// TIA Portal V21 export
ORGANIZATION_BLOCK "Date_Time_Block"   // OB200, LAD, ProgramCycle
{ S7_Optimized_Access := 'TRUE' }
// stored: SetENOAutomatically false
   VAR_TEMP   // added for the SCL form of the ladder/FBD networks
      _w1 : Bool;
      _w2 : Bool;
      _w3 : Bool;
   END_VAR
BEGIN

REGION Network 1: Convert Date to String
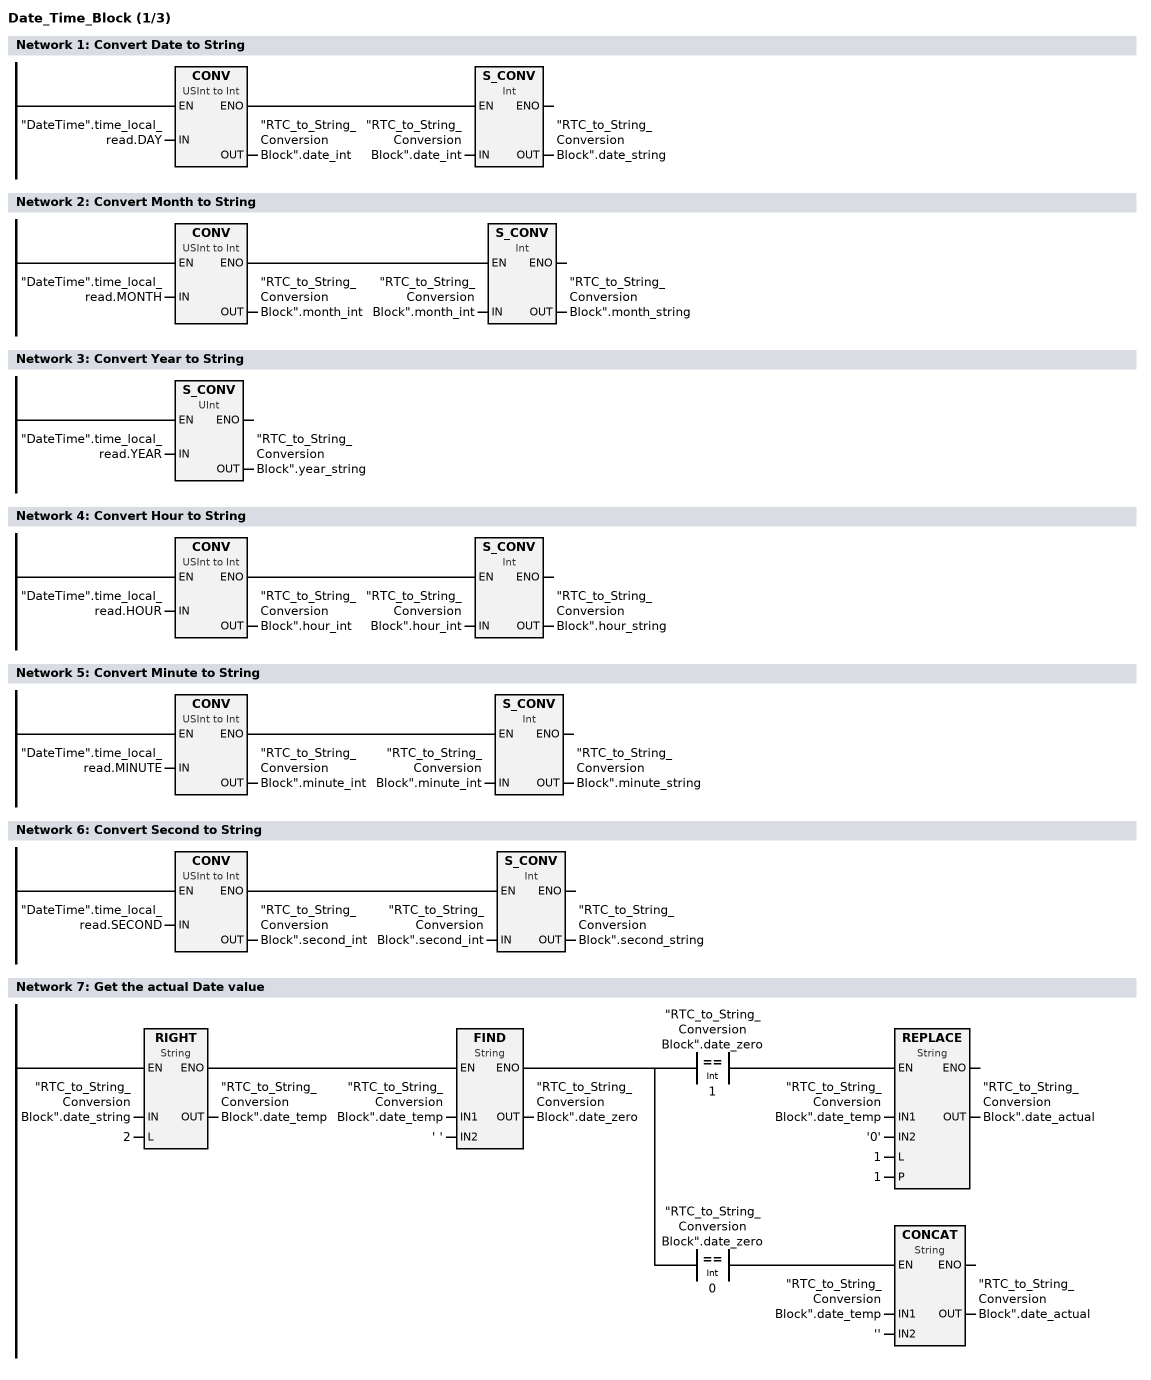
   RUNG wire#powerrail
      { S7_Templates := "[SrcType := USInt, DestType := Int]"; S7_GenerateENO := "TRUE" } Convert(in := "DateTime".time_local_read.DAY, out => "RTC_to_String_Conversion Block".date_int)
      { S7_Templates := "[src_type := Int, dest_type := String]" } S_CONV(IN := "RTC_to_String_Conversion Block".date_int, OUT => "RTC_to_String_Conversion Block".date_string)
   END_RUNG
   // the same network as SCL:
   // ENO of a box is taken as its EN; it also drops when the box reports an error
   "RTC_to_String_Conversion Block".date_int := USINT_TO_INT("DateTime".time_local_read.DAY);
   S_CONV(IN := "RTC_to_String_Conversion Block".date_int, OUT => "RTC_to_String_Conversion Block".date_string);
END_REGION

REGION Network 2: Convert Month to String
   RUNG wire#powerrail
      { S7_Templates := "[SrcType := USInt, DestType := Int]"; S7_GenerateENO := "TRUE" } Convert(in := "DateTime".time_local_read.MONTH, out => "RTC_to_String_Conversion Block".month_int)
      { S7_Templates := "[src_type := Int, dest_type := String]" } S_CONV(IN := "RTC_to_String_Conversion Block".month_int, OUT => "RTC_to_String_Conversion Block".month_string)
   END_RUNG
   // the same network as SCL:
   // ENO of a box is taken as its EN; it also drops when the box reports an error
   "RTC_to_String_Conversion Block".month_int := USINT_TO_INT("DateTime".time_local_read.MONTH);
   S_CONV(IN := "RTC_to_String_Conversion Block".month_int,
          OUT => "RTC_to_String_Conversion Block".month_string);
END_REGION

REGION Network 3: Convert Year to String
   RUNG wire#powerrail
      { S7_Templates := "[src_type := UInt, dest_type := String]" } S_CONV(IN := "DateTime".time_local_read.YEAR, OUT => "RTC_to_String_Conversion Block".year_string)
   END_RUNG
   // the same network as SCL:
   S_CONV(IN := "DateTime".time_local_read.YEAR, OUT => "RTC_to_String_Conversion Block".year_string);
END_REGION

REGION Network 4: Convert Hour to String
   RUNG wire#powerrail
      { S7_Templates := "[SrcType := USInt, DestType := Int]"; S7_GenerateENO := "TRUE" } Convert(in := "DateTime".time_local_read.HOUR, out => "RTC_to_String_Conversion Block".hour_int)
      { S7_Templates := "[src_type := Int, dest_type := String]" } S_CONV(IN := "RTC_to_String_Conversion Block".hour_int, OUT => "RTC_to_String_Conversion Block".hour_string)
   END_RUNG
   // the same network as SCL:
   // ENO of a box is taken as its EN; it also drops when the box reports an error
   "RTC_to_String_Conversion Block".hour_int := USINT_TO_INT("DateTime".time_local_read.HOUR);
   S_CONV(IN := "RTC_to_String_Conversion Block".hour_int, OUT => "RTC_to_String_Conversion Block".hour_string);
END_REGION

REGION Network 5: Convert Minute to String
   RUNG wire#powerrail
      { S7_Templates := "[SrcType := USInt, DestType := Int]"; S7_GenerateENO := "TRUE" } Convert(in := "DateTime".time_local_read.MINUTE, out => "RTC_to_String_Conversion Block".minute_int)
      { S7_Templates := "[src_type := Int, dest_type := String]" } S_CONV(IN := "RTC_to_String_Conversion Block".minute_int, OUT => "RTC_to_String_Conversion Block".minute_string)
   END_RUNG
   // the same network as SCL:
   // ENO of a box is taken as its EN; it also drops when the box reports an error
   "RTC_to_String_Conversion Block".minute_int := USINT_TO_INT("DateTime".time_local_read.MINUTE);
   S_CONV(IN := "RTC_to_String_Conversion Block".minute_int,
          OUT => "RTC_to_String_Conversion Block".minute_string);
END_REGION

REGION Network 6: Convert Second to String
   RUNG wire#powerrail
      { S7_Templates := "[SrcType := USInt, DestType := Int]"; S7_GenerateENO := "TRUE" } Convert(in := "DateTime".time_local_read.SECOND, out => "RTC_to_String_Conversion Block".second_int)
      { S7_Templates := "[src_type := Int, dest_type := String]" } S_CONV(IN := "RTC_to_String_Conversion Block".second_int, OUT => "RTC_to_String_Conversion Block".second_string)
   END_RUNG
   // the same network as SCL:
   // ENO of a box is taken as its EN; it also drops when the box reports an error
   "RTC_to_String_Conversion Block".second_int := USINT_TO_INT("DateTime".time_local_read.SECOND);
   S_CONV(IN := "RTC_to_String_Conversion Block".second_int,
          OUT => "RTC_to_String_Conversion Block".second_string);
END_REGION

REGION Network 7: Get the actual Date value
   RUNG wire#powerrail
      { S7_Templates := "str_type := String" } RIGHT(IN := "RTC_to_String_Conversion Block".date_string, L := 2, OUT => "RTC_to_String_Conversion Block".date_temp)
      { S7_Templates := "str_type := String" } FIND(IN1 := "RTC_to_String_Conversion Block".date_temp, IN2 := ' ', OUT => "RTC_to_String_Conversion Block".date_zero)
      wire#w1
      { S7_Templates := "SrcType := Int" } EQ_Contact(in1 := "RTC_to_String_Conversion Block".date_zero, in2 := 1)
      { S7_Templates := "str_type := String" } REPLACE(IN1 := "RTC_to_String_Conversion Block".date_temp, IN2 := '0', L := 1, P := 1, OUT => "RTC_to_String_Conversion Block".date_actual)
   END_RUNG
   RUNG wire#w1
      { S7_Templates := "SrcType := Int" } EQ_Contact(in1 := "RTC_to_String_Conversion Block".date_zero, in2 := 0)
      { S7_Templates := "[card := 2, str_type := String]" } CONCAT(IN1 := "RTC_to_String_Conversion Block".date_temp, IN2 := '', OUT => "RTC_to_String_Conversion Block".date_actual)
   END_RUNG
   // the same network as SCL:
   RIGHT(IN := "RTC_to_String_Conversion Block".date_string,
         L := 2,
         OUT => "RTC_to_String_Conversion Block".date_temp,
         ENO => #_w1);
   FIND(EN := #_w1,
        IN1 := "RTC_to_String_Conversion Block".date_temp,
        IN2 := ' ',
        OUT => "RTC_to_String_Conversion Block".date_zero,
        ENO => #_w2);
   IF #_w2 AND ("RTC_to_String_Conversion Block".date_zero = 1) THEN
       REPLACE(IN1 := "RTC_to_String_Conversion Block".date_temp,
               IN2 := '0',
               L := 1,
               P := 1,
               OUT => "RTC_to_String_Conversion Block".date_actual);
   END_IF;
   IF #_w2 AND ("RTC_to_String_Conversion Block".date_zero = 0) THEN
       CONCAT(IN1 := "RTC_to_String_Conversion Block".date_temp,
              IN2 := '',
              OUT => "RTC_to_String_Conversion Block".date_actual);
   END_IF;
END_REGION

REGION Network 8: Get the actual month value
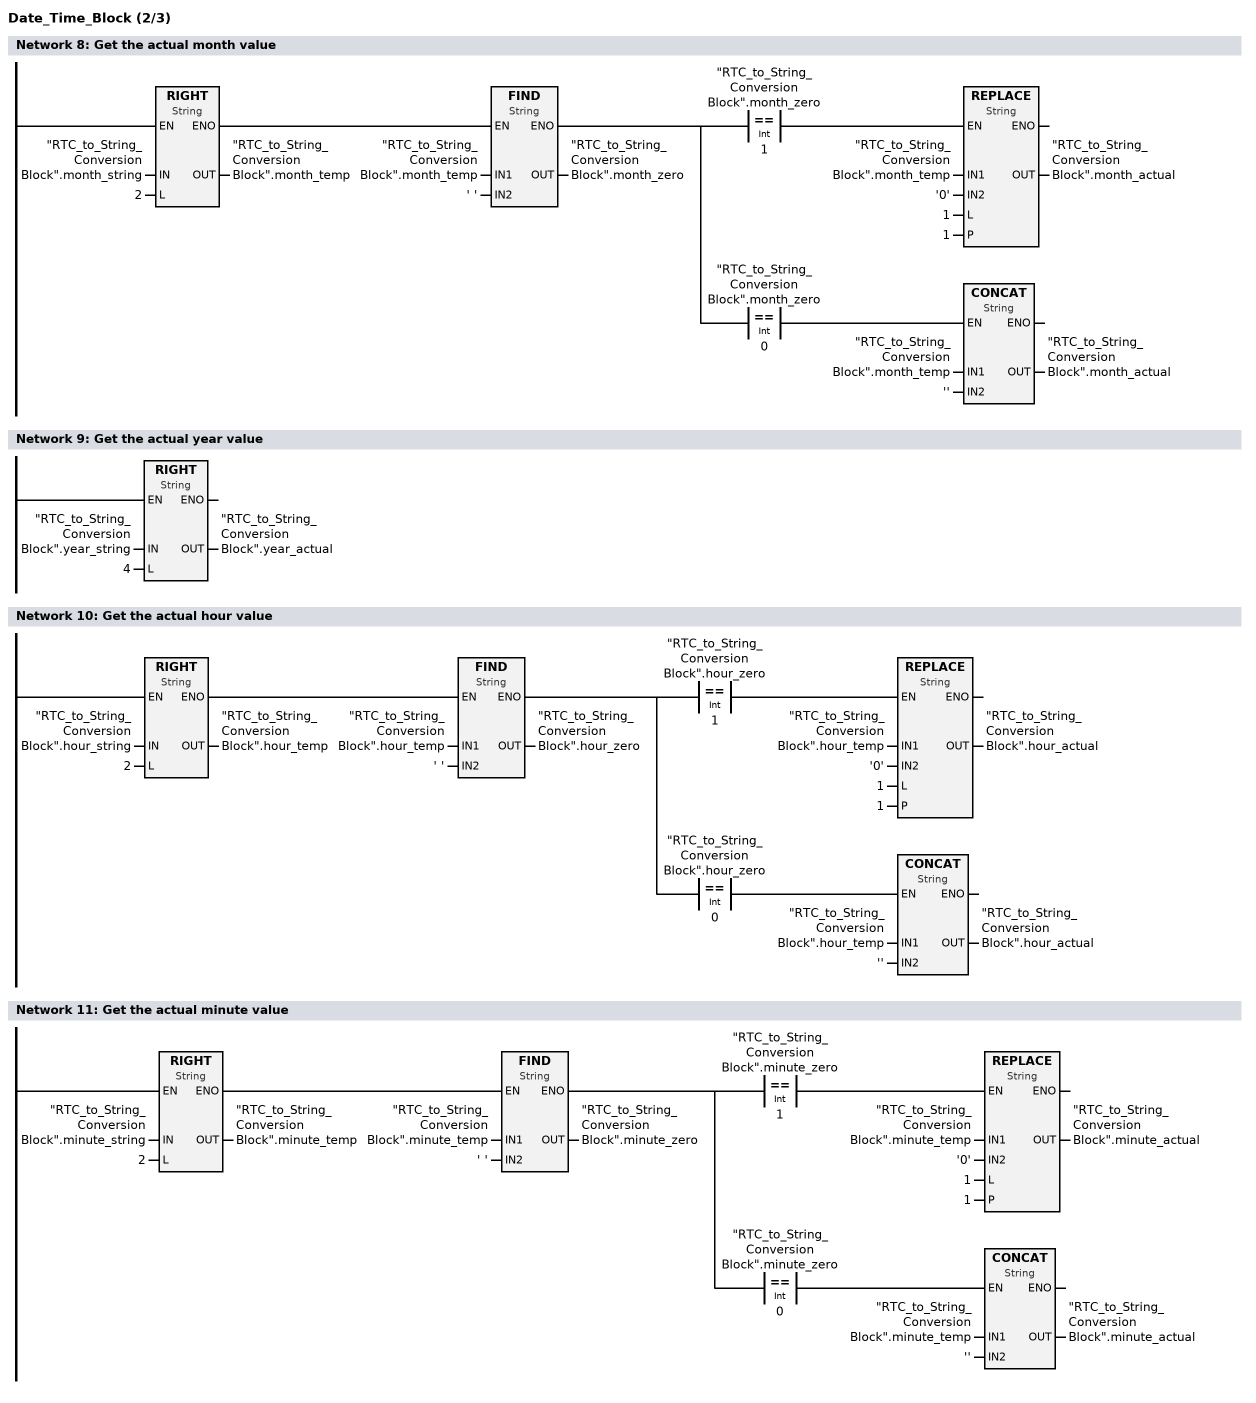
   RUNG wire#powerrail
      { S7_Templates := "str_type := String" } RIGHT(IN := "RTC_to_String_Conversion Block".month_string, L := 2, OUT => "RTC_to_String_Conversion Block".month_temp)
      { S7_Templates := "str_type := String" } FIND(IN1 := "RTC_to_String_Conversion Block".month_temp, IN2 := ' ', OUT => "RTC_to_String_Conversion Block".month_zero)
      wire#w1
      { S7_Templates := "SrcType := Int" } EQ_Contact(in1 := "RTC_to_String_Conversion Block".month_zero, in2 := 1)
      { S7_Templates := "str_type := String" } REPLACE(IN1 := "RTC_to_String_Conversion Block".month_temp, IN2 := '0', L := 1, P := 1, OUT => "RTC_to_String_Conversion Block".month_actual)
   END_RUNG
   RUNG wire#w1
      { S7_Templates := "SrcType := Int" } EQ_Contact(in1 := "RTC_to_String_Conversion Block".month_zero, in2 := 0)
      { S7_Templates := "[card := 2, str_type := String]" } CONCAT(IN1 := "RTC_to_String_Conversion Block".month_temp, IN2 := '', OUT => "RTC_to_String_Conversion Block".month_actual)
   END_RUNG
   // the same network as SCL:
   RIGHT(IN := "RTC_to_String_Conversion Block".month_string,
         L := 2,
         OUT => "RTC_to_String_Conversion Block".month_temp,
         ENO => #_w1);
   FIND(EN := #_w1,
        IN1 := "RTC_to_String_Conversion Block".month_temp,
        IN2 := ' ',
        OUT => "RTC_to_String_Conversion Block".month_zero,
        ENO => #_w2);
   IF #_w2 AND ("RTC_to_String_Conversion Block".month_zero = 1) THEN
       REPLACE(IN1 := "RTC_to_String_Conversion Block".month_temp,
               IN2 := '0',
               L := 1,
               P := 1,
               OUT => "RTC_to_String_Conversion Block".month_actual);
   END_IF;
   IF #_w2 AND ("RTC_to_String_Conversion Block".month_zero = 0) THEN
       CONCAT(IN1 := "RTC_to_String_Conversion Block".month_temp,
              IN2 := '',
              OUT => "RTC_to_String_Conversion Block".month_actual);
   END_IF;
END_REGION

REGION Network 9: Get the actual year value
   RUNG wire#powerrail
      { S7_Templates := "str_type := String" } RIGHT(IN := "RTC_to_String_Conversion Block".year_string, L := 4, OUT => "RTC_to_String_Conversion Block".year_actual)
   END_RUNG
   // the same network as SCL:
   RIGHT(IN := "RTC_to_String_Conversion Block".year_string,
         L := 4,
         OUT => "RTC_to_String_Conversion Block".year_actual);
END_REGION

REGION Network 10: Get the actual hour value
   RUNG wire#powerrail
      { S7_Templates := "str_type := String" } RIGHT(IN := "RTC_to_String_Conversion Block".hour_string, L := 2, OUT => "RTC_to_String_Conversion Block".hour_temp)
      { S7_Templates := "str_type := String" } FIND(IN1 := "RTC_to_String_Conversion Block".hour_temp, IN2 := ' ', OUT => "RTC_to_String_Conversion Block".hour_zero)
      wire#w1
      { S7_Templates := "SrcType := Int" } EQ_Contact(in1 := "RTC_to_String_Conversion Block".hour_zero, in2 := 1)
      { S7_Templates := "str_type := String" } REPLACE(IN1 := "RTC_to_String_Conversion Block".hour_temp, IN2 := '0', L := 1, P := 1, OUT => "RTC_to_String_Conversion Block".hour_actual)
   END_RUNG
   RUNG wire#w1
      { S7_Templates := "SrcType := Int" } EQ_Contact(in1 := "RTC_to_String_Conversion Block".hour_zero, in2 := 0)
      { S7_Templates := "[card := 2, str_type := String]" } CONCAT(IN1 := "RTC_to_String_Conversion Block".hour_temp, IN2 := '', OUT => "RTC_to_String_Conversion Block".hour_actual)
   END_RUNG
   // the same network as SCL:
   RIGHT(IN := "RTC_to_String_Conversion Block".hour_string,
         L := 2,
         OUT => "RTC_to_String_Conversion Block".hour_temp,
         ENO => #_w1);
   FIND(EN := #_w1,
        IN1 := "RTC_to_String_Conversion Block".hour_temp,
        IN2 := ' ',
        OUT => "RTC_to_String_Conversion Block".hour_zero,
        ENO => #_w2);
   IF #_w2 AND ("RTC_to_String_Conversion Block".hour_zero = 1) THEN
       REPLACE(IN1 := "RTC_to_String_Conversion Block".hour_temp,
               IN2 := '0',
               L := 1,
               P := 1,
               OUT => "RTC_to_String_Conversion Block".hour_actual);
   END_IF;
   IF #_w2 AND ("RTC_to_String_Conversion Block".hour_zero = 0) THEN
       CONCAT(IN1 := "RTC_to_String_Conversion Block".hour_temp,
              IN2 := '',
              OUT => "RTC_to_String_Conversion Block".hour_actual);
   END_IF;
END_REGION

REGION Network 11: Get the actual minute value
   RUNG wire#powerrail
      { S7_Templates := "str_type := String" } RIGHT(IN := "RTC_to_String_Conversion Block".minute_string, L := 2, OUT => "RTC_to_String_Conversion Block".minute_temp)
      { S7_Templates := "str_type := String" } FIND(IN1 := "RTC_to_String_Conversion Block".minute_temp, IN2 := ' ', OUT => "RTC_to_String_Conversion Block".minute_zero)
      wire#w1
      { S7_Templates := "SrcType := Int" } EQ_Contact(in1 := "RTC_to_String_Conversion Block".minute_zero, in2 := 1)
      { S7_Templates := "str_type := String" } REPLACE(IN1 := "RTC_to_String_Conversion Block".minute_temp, IN2 := '0', L := 1, P := 1, OUT => "RTC_to_String_Conversion Block".minute_actual)
   END_RUNG
   RUNG wire#w1
      { S7_Templates := "SrcType := Int" } EQ_Contact(in1 := "RTC_to_String_Conversion Block".minute_zero, in2 := 0)
      { S7_Templates := "[card := 2, str_type := String]" } CONCAT(IN1 := "RTC_to_String_Conversion Block".minute_temp, IN2 := '', OUT => "RTC_to_String_Conversion Block".minute_actual)
   END_RUNG
   // the same network as SCL:
   RIGHT(IN := "RTC_to_String_Conversion Block".minute_string,
         L := 2,
         OUT => "RTC_to_String_Conversion Block".minute_temp,
         ENO => #_w1);
   FIND(EN := #_w1,
        IN1 := "RTC_to_String_Conversion Block".minute_temp,
        IN2 := ' ',
        OUT => "RTC_to_String_Conversion Block".minute_zero,
        ENO => #_w2);
   IF #_w2 AND ("RTC_to_String_Conversion Block".minute_zero = 1) THEN
       REPLACE(IN1 := "RTC_to_String_Conversion Block".minute_temp,
               IN2 := '0',
               L := 1,
               P := 1,
               OUT => "RTC_to_String_Conversion Block".minute_actual);
   END_IF;
   IF #_w2 AND ("RTC_to_String_Conversion Block".minute_zero = 0) THEN
       CONCAT(IN1 := "RTC_to_String_Conversion Block".minute_temp,
              IN2 := '',
              OUT => "RTC_to_String_Conversion Block".minute_actual);
   END_IF;
END_REGION

REGION Network 12: Get the actual second value
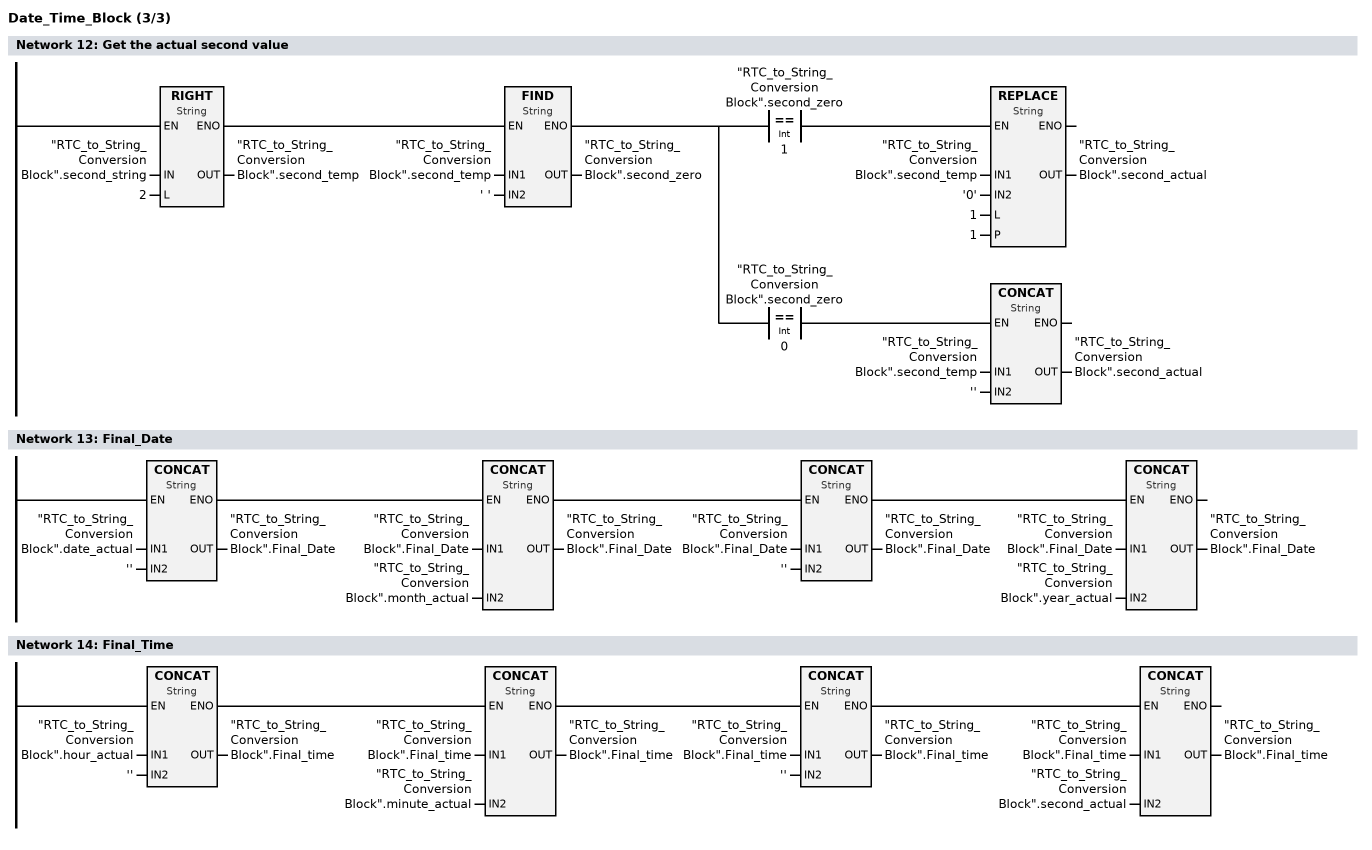
   RUNG wire#powerrail
      { S7_Templates := "str_type := String" } RIGHT(IN := "RTC_to_String_Conversion Block".second_string, L := 2, OUT => "RTC_to_String_Conversion Block".second_temp)
      { S7_Templates := "str_type := String" } FIND(IN1 := "RTC_to_String_Conversion Block".second_temp, IN2 := ' ', OUT => "RTC_to_String_Conversion Block".second_zero)
      wire#w1
      { S7_Templates := "SrcType := Int" } EQ_Contact(in1 := "RTC_to_String_Conversion Block".second_zero, in2 := 1)
      { S7_Templates := "str_type := String" } REPLACE(IN1 := "RTC_to_String_Conversion Block".second_temp, IN2 := '0', L := 1, P := 1, OUT => "RTC_to_String_Conversion Block".second_actual)
   END_RUNG
   RUNG wire#w1
      { S7_Templates := "SrcType := Int" } EQ_Contact(in1 := "RTC_to_String_Conversion Block".second_zero, in2 := 0)
      { S7_Templates := "[card := 2, str_type := String]" } CONCAT(IN1 := "RTC_to_String_Conversion Block".second_temp, IN2 := '', OUT => "RTC_to_String_Conversion Block".second_actual)
   END_RUNG
   // the same network as SCL:
   RIGHT(IN := "RTC_to_String_Conversion Block".second_string,
         L := 2,
         OUT => "RTC_to_String_Conversion Block".second_temp,
         ENO => #_w1);
   FIND(EN := #_w1,
        IN1 := "RTC_to_String_Conversion Block".second_temp,
        IN2 := ' ',
        OUT => "RTC_to_String_Conversion Block".second_zero,
        ENO => #_w2);
   IF #_w2 AND ("RTC_to_String_Conversion Block".second_zero = 1) THEN
       REPLACE(IN1 := "RTC_to_String_Conversion Block".second_temp,
               IN2 := '0',
               L := 1,
               P := 1,
               OUT => "RTC_to_String_Conversion Block".second_actual);
   END_IF;
   IF #_w2 AND ("RTC_to_String_Conversion Block".second_zero = 0) THEN
       CONCAT(IN1 := "RTC_to_String_Conversion Block".second_temp,
              IN2 := '',
              OUT => "RTC_to_String_Conversion Block".second_actual);
   END_IF;
END_REGION

REGION Network 13: Final_Date
   RUNG wire#powerrail
      { S7_Templates := "[card := 2, str_type := String]" } CONCAT(IN1 := "RTC_to_String_Conversion Block".date_actual, IN2 := '', OUT => "RTC_to_String_Conversion Block".Final_Date)
      { S7_Templates := "[card := 2, str_type := String]" } CONCAT(IN1 := "RTC_to_String_Conversion Block".Final_Date, IN2 := "RTC_to_String_Conversion Block".month_actual, OUT => "RTC_to_String_Conversion Block".Final_Date)
      { S7_Templates := "[card := 2, str_type := String]" } CONCAT(IN1 := "RTC_to_String_Conversion Block".Final_Date, IN2 := '', OUT => "RTC_to_String_Conversion Block".Final_Date)
      { S7_Templates := "[card := 2, str_type := String]" } CONCAT(IN1 := "RTC_to_String_Conversion Block".Final_Date, IN2 := "RTC_to_String_Conversion Block".year_actual, OUT => "RTC_to_String_Conversion Block".Final_Date)
   END_RUNG
   // the same network as SCL:
   CONCAT(IN1 := "RTC_to_String_Conversion Block".date_actual,
          IN2 := '',
          OUT => "RTC_to_String_Conversion Block".Final_Date,
          ENO => #_w1);
   CONCAT(EN := #_w1,
          IN1 := "RTC_to_String_Conversion Block".Final_Date,
          IN2 := "RTC_to_String_Conversion Block".month_actual,
          OUT => "RTC_to_String_Conversion Block".Final_Date,
          ENO => #_w2);
   CONCAT(EN := #_w2,
          IN1 := "RTC_to_String_Conversion Block".Final_Date,
          IN2 := '',
          OUT => "RTC_to_String_Conversion Block".Final_Date,
          ENO => #_w3);
   IF #_w3 THEN
       CONCAT(IN1 := "RTC_to_String_Conversion Block".Final_Date,
              IN2 := "RTC_to_String_Conversion Block".year_actual,
              OUT => "RTC_to_String_Conversion Block".Final_Date);
   END_IF;
END_REGION

REGION Network 14: Final_Time
   RUNG wire#powerrail
      { S7_Templates := "[card := 2, str_type := String]" } CONCAT(IN1 := "RTC_to_String_Conversion Block".hour_actual, IN2 := '', OUT => "RTC_to_String_Conversion Block".Final_time)
      { S7_Templates := "[card := 2, str_type := String]" } CONCAT(IN1 := "RTC_to_String_Conversion Block".Final_time, IN2 := "RTC_to_String_Conversion Block".minute_actual, OUT => "RTC_to_String_Conversion Block".Final_time)
      { S7_Templates := "[card := 2, str_type := String]" } CONCAT(IN1 := "RTC_to_String_Conversion Block".Final_time, IN2 := '', OUT => "RTC_to_String_Conversion Block".Final_time)
      { S7_Templates := "[card := 2, str_type := String]" } CONCAT(IN1 := "RTC_to_String_Conversion Block".Final_time, IN2 := "RTC_to_String_Conversion Block".second_actual, OUT => "RTC_to_String_Conversion Block".Final_time)
   END_RUNG
   // the same network as SCL:
   CONCAT(IN1 := "RTC_to_String_Conversion Block".hour_actual,
          IN2 := '',
          OUT => "RTC_to_String_Conversion Block".Final_time,
          ENO => #_w1);
   CONCAT(EN := #_w1,
          IN1 := "RTC_to_String_Conversion Block".Final_time,
          IN2 := "RTC_to_String_Conversion Block".minute_actual,
          OUT => "RTC_to_String_Conversion Block".Final_time,
          ENO => #_w2);
   CONCAT(EN := #_w2,
          IN1 := "RTC_to_String_Conversion Block".Final_time,
          IN2 := '',
          OUT => "RTC_to_String_Conversion Block".Final_time,
          ENO => #_w3);
   IF #_w3 THEN
       CONCAT(IN1 := "RTC_to_String_Conversion Block".Final_time,
              IN2 := "RTC_to_String_Conversion Block".second_actual,
              OUT => "RTC_to_String_Conversion Block".Final_time);
   END_IF;
END_REGION
END_ORGANIZATION_BLOCK
